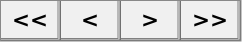
VISUALIZATION V_NumInputReal  // 242x42
VAR_INPUT
	INrValueMin		: REAL;
	INrValueMax		: REAL;
	INrStepMin		: REAL;
	INrStepMax		: REAL;
END_VAR
VAR_IN_OUT
	INrVariable		: REAL;
END_VAR
    Button (120,0 60x40), ">", invisible if: INrVariable >= INrValueMax
        OnMouseClick: execute {
            INrVariable :=
            	INrVariable
            	+ INrStepMin;
        }
    Button (60,0 60x40), "<", invisible if: INrVariable <= INrValueMin
        OnMouseClick: execute {
            INrVariable :=
            	INrVariable
            	- INrStepMin;
        }
    Button (180,0 60x40), ">>", invisible if: INrVariable >= INrValueMax
        OnMouseClick: execute {
            INrVariable :=
            	INrVariable
            	+ INrStepMax;
        }
    Button (0,0 60x40), "<<", invisible if: INrVariable <= INrValueMin
        OnMouseClick: execute {
            INrVariable :=
            	INrVariable
            	- INrStepMax;
        }
END_VISUALIZATION

(* stored: Version 1.1.0.1, ProductVersion 3.1.4018.5
   Visu V_NumInputReal: Id {0c6b8483-457e-4ae4-b590-38caa1fd09d3} *)
